(* PLC project LD_EVOLUTION_6, Beckhoff Automation GmbH TwinCAT PLC Control 3.5.10.30 *)
(* stored: creationDateTime 2019-09-26T16:29:19.1573185, modificationDateTime 2019-09-26T16:29:19.1573185 *)

PROGRAM Main
VAR
	A: BOOL;
	B: BOOL;
	Open: BOOL;
	C: BOOL;
	Count: BOOL;
END_VAR
  VAR  (* added by the conversion: wires and edge detectors of the diagram *)
    _EXECUTE3_EN : BOOL;
  END_VAR

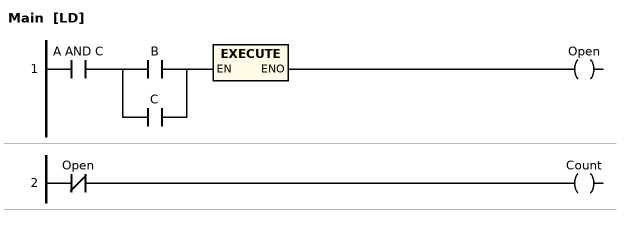
(* LD diagram, written out as Structured Text *)

_EXECUTE3_EN := (A AND C) AND (B OR C);
IF _EXECUTE3_EN THEN
  C:= A AND B;
  Open := C;
END_IF;
Open := _EXECUTE3_EN;

Count := NOT Open;
END_PROGRAM

CONFIGURATION Application
  RESOURCE LD_EVOLUTION_6 ON PLC
(* global variable list GVL *)
{attribute 'qualified_only'}
VAR_GLOBAL
	IsSFCResetting : BOOL;
END_VAR
    TASK PlcTask(INTERVAL := T#0ms, PRIORITY := 20);
    PROGRAM Main WITH PlcTask : Main;
  END_RESOURCE
END_CONFIGURATION
